TYPE ACRMemoryLRealEvent EXTENDS ACRMemoryEvent :
STRUCT
	_Value : LREAL;
END_STRUCT
END_TYPE

(* stored: Version 1.1.0.1, ProductVersion 3.1.4020.12
   DUT ACRMemoryLRealEvent: Id {4ac6a87a-456f-496e-a1e0-c1578db3020d} *)
